(* CoDeSys 2.3.9.62 project: Practica1Ej1.pro *)
(* Libraries: Standard.lib 4.10.05 11:14:46, IecSfc.lib 2.6.14 10:37:46 *)

(* Global variable list: Global_Variables *)
VAR_GLOBAL
     (* Variables de entrada *)
      START:BOOL;
	A:BOOL;
	B:BOOL;
      CC:BOOL;  (*Botón para comienzo de carga*)
      FC:BOOL;   (*Botçon para fin de carga *)
      (* Variables de salida *)
	MOTOR_IZ:BOOL;
	MOTOR_DE:BOOL;
      Carga:BOOL;

       (* Variables para la simulación *)
	Vel:INT:=1;
END_VAR

(* POU PLC_PRG, FBD *)
PROGRAM PLC_PRG
VAR

END_VAR
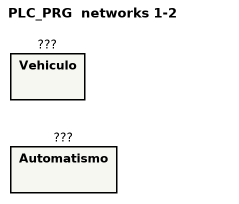
_FBD_ (* Function Block Diagram *)
NETWORK 1
	???:Vehiculo()
NETWORK 2
	???:Automatismo()
_END_FBD_
END_PROGRAM

(* POU Vehiculo, ST *)
PROGRAM Vehiculo
VAR
	PosX: INT;
END_VAR
A:=FALSE;
B:=FALSE;


IF MOTOR_DE=TRUE THEN

     PosX:=PosX+Vel;

END_IF

IF MOTOR_IZ=TRUE THEN

     PosX:=PosX-Vel;

END_IF


IF PosX<=0 THEN
   A:=TRUE;
END_IF

IF PosX>=400 THEN
  B:=TRUE;
END_IF
END_PROGRAM

(* POU Automatismo, LD *)
PROGRAM Automatismo
VAR

	E0: BOOL;
	E1: BOOL;
	E2: BOOL;
	E3: BOOL;
	E4: BOOL;
END_VAR
VAR (* helpers for the ST form of the networks *)
	_p1 : BOOL;
	_p2 : BOOL;
	_p3 : BOOL;
	_p4 : BOOL;
	_p5 : BOOL;
END_VAR
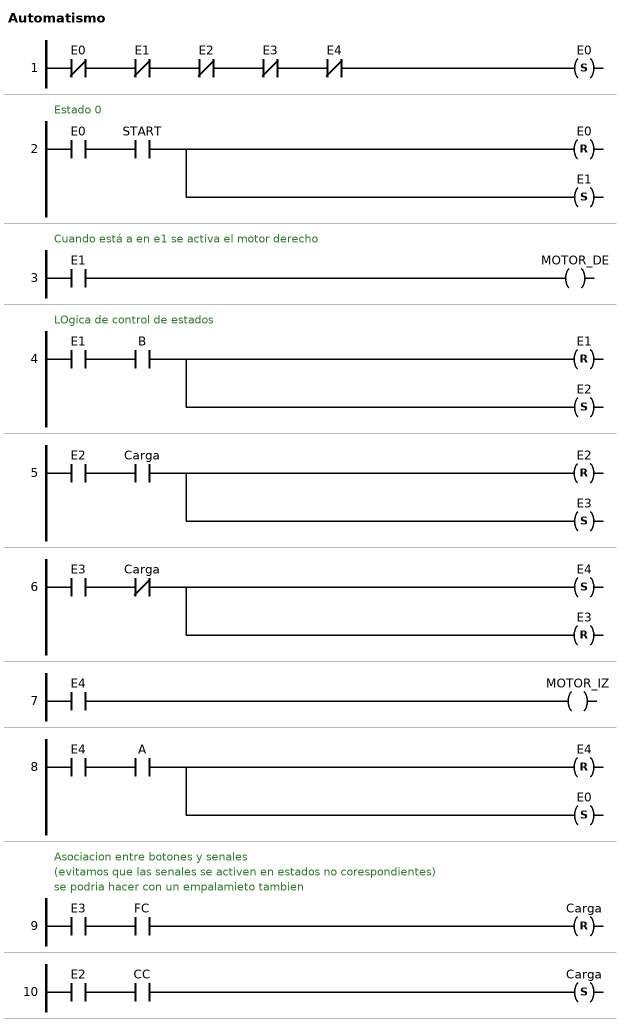
_LD_ (* Ladder Diagram *)
NETWORK 1
	[/E0] - [/E1] - [/E2] - [/E3] - [/E4] --- (S E0)
NETWORK 2 (* Estado 0 *)
	[E0] - [START] --- (R E0) (S E1)
NETWORK 3 (* Cuando está a en e1 se activa el motor derecho *)
	[E1] --- (MOTOR_DE)
NETWORK 4 (* LOgica de control de estados *)
	[E1] - [B] --- (R E1) (S E2)
NETWORK 5
	[E2] - [Carga] --- (R E2) (S E3)
NETWORK 6
	[E3] - [/Carga] --- (S E4) (R E3)
NETWORK 7
	[E4] --- (MOTOR_IZ)
NETWORK 8
	[E4] - [A] --- (R E4) (S E0)
NETWORK 9 (* Asociacion entre botones y senales / (evitamos que las senales se activen en estados no corespondientes) / se podria hacer con un empalamieto tambien *)
	[E3] - [FC] --- (R Carga)
NETWORK 10
	[E2] - [CC] --- (S Carga)
_END_LD_
(* the same logic as Structured Text *)
(* Network 1 *)
IF NOT E0 AND NOT E1 AND NOT E2 AND NOT E3 AND NOT E4 THEN E0 := TRUE; END_IF;
(* Network 2: Estado 0 *)
_p1 := E0 AND START;
IF _p1 THEN E0 := FALSE; E1 := TRUE; END_IF;
(* Network 3: Cuando está a en e1 se activa el motor derecho *)
MOTOR_DE := E1;
(* Network 4: LOgica de control de estados *)
_p2 := E1 AND B;
IF _p2 THEN E1 := FALSE; E2 := TRUE; END_IF;
(* Network 5 *)
_p3 := E2 AND Carga;
IF _p3 THEN E2 := FALSE; E3 := TRUE; END_IF;
(* Network 6 *)
_p4 := E3 AND NOT Carga;
IF _p4 THEN E4 := TRUE; E3 := FALSE; END_IF;
(* Network 7 *)
MOTOR_IZ := E4;
(* Network 8 *)
_p5 := E4 AND A;
IF _p5 THEN E4 := FALSE; E0 := TRUE; END_IF;
(* Network 9: Asociacion entre botones y senales / (evitamos que las senales se activen en estados no corespondientes) / se podria hacer con un empalamieto tambien *)
IF E3 AND FC THEN Carga := FALSE; END_IF;
(* Network 10 *)
IF E2 AND CC THEN Carga := TRUE; END_IF;
END_PROGRAM

(* Visualisation Vehiculo
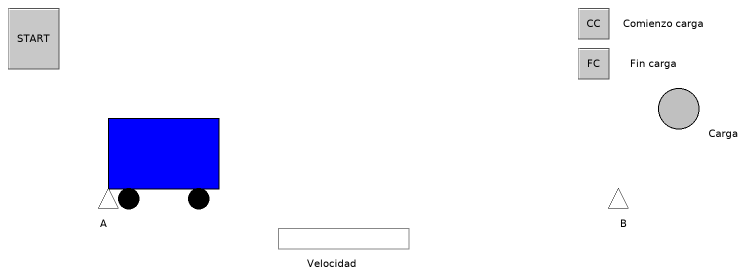
rectangle at (140,120)-(251,191): x offset Vehiculo.PosX
polygon at (130,190)-(150,210): alarm colour if .A
polygon at (640,190)-(660,210): alarm colour if .B
button at (40,10)-(91,71): text "START"; taps START
ellipse at (150,190)-(171,211): x offset Vehiculo.PosX
ellipse at (220,190)-(241,211): x offset Vehiculo.PosX
rectangle at (310,250)-(421,281): text "Velocidad"
rectangle at (80,210)-(191,241): text "A"
rectangle at (600,210)-(711,241): text "B"
button at (610,10)-(641,41): text "CC"; taps CC
button at (610,50)-(641,81): text "FC"; taps FC
ellipse at (690,90)-(731,131): alarm colour if Carga
rectangle at (640,10)-(751,41): text "Comienzo carga"
rectangle at (650,50)-(721,81): text "Fin carga"
rectangle at (700,120)-(811,151): text "Carga"
1 more shapes without text or variables
*)
